FUNCTION_BLOCK FB_CRYO_VALVE_CTRL EXTENDS FB_CRYO_BIN_CTRL
VAR_INPUT
END_VAR
VAR_OUTPUT
END_VAR
VAR
	//
	// Alarm handling
	//
	// List of alarms to be handled by Valve.
	// Alarms cannot be defined in FB_CRYO_BIN_CTRL,
	// because they are specific to the device/controller.
	// There are three alarms for Valves:
	//   0: NOT_OP
	//   1: CLOSE failed
	//   2: OPEN  failed
	arrEventEntry : ARRAY [0..2] OF TcEventEntry;
	// Alarm handler FB
	fbAlarmHandler : FB_AlarmHandler;
END_VAR

// This call just configures logs at the very start.
// Logging is done by explicit calls to M_LogInfo().
logs(in_sName := in_sName);


// Execute parent FB.
SUPER^();


// Update the status.
// This will handle alarms as well.
M_SetStatus(stat.nState);

METHOD M_Configure
VAR_INPUT
END_VAR
// Device specific implementation
// 
arrEventEntry[0] := Tc_Events.CryoValveEventClass.HardwareError;
arrEventEntry[1] := Tc_Events.CryoValveEventClass.FailureOpen;
arrEventEntry[2] := Tc_Events.CryoValveEventClass.FailureClose;


// A MUST !!!
stat.bConfigured	:= TRUE;
END_METHOD

//
// Overrides the same method in FB_CRYO_BIN_CTRL.
//
// Set labels for logging.
//	OPEN, CLOSE (for valves)
METHOD M_GetStateLabel : STRING
VAR_INPUT
	state:	E_CRYO_BIN_CTRL_STATE;
END_VAR
CASE state OF
	E_CRYO_BIN_CTRL_STATE.OFF:
		M_GetStateLabel	:= 'CLOSED';
	
	E_CRYO_BIN_CTRL_STATE.ACTIVE_SWITCHING_ON:
		M_GetStateLabel	:= 'OPENING...';
	
	E_CRYO_BIN_CTRL_STATE.ACTIVE_OFF:
		M_GetStateLabel	:= 'CLOSED';
	
	E_CRYO_BIN_CTRL_STATE.ACTIVE_ON:
		M_GetStateLabel	:= 'OPEN';
	
	E_CRYO_BIN_CTRL_STATE.ACTIVE_SWITCHING_OFF:
		M_GetStateLabel	:= 'CLOSING...';
	
	E_CRYO_BIN_CTRL_STATE.ERROR:
		M_GetStateLabel	:= 'ERROR';
END_CASE
END_METHOD

METHOD M_SetStatus
VAR_INPUT
	nState:	E_CRYO_BIN_CTRL_STATE;
END_VAR
// Execute the status of the parent FB.
SUPER^.M_SetStatus(nState);


// Handle alarms
M_UpdateAlarms();
END_METHOD

METHOD M_UpdateAlarms
VAR_INPUT
END_VAR
VAR
	stEventEntry : TcEventEntry;
	sText : STRING;
END_VAR
// Array of EventEntry is initialised in the M_Configure method with 
// the alarms defined for the Valve.

fbAlarmHandler(stAlarms := stat.stAlarms);


// Trigger alarms in case of failure.
// The alarms are raised with a rising edge trigger.
// The alarms are cleared with a falling edge trigger.
IF stat.nState = E_CRYO_BIN_CTRL_STATE.ERROR THEN
	IF Actuator.i_nCouplerState <> 8 THEN
		// System not OPERATIONAL or
		// i_nCouplerState not linked to State variable.
		fbAlarmHandler.M_SetAlarm(Tc_Events.CryoValveEventClass.HardwareError);
		stat.sState	:= 'ERROR: System not OPERATIONAL';
	ELSIF Actuator.stat.nLastCommand = E_CRYO_BIN_ACT_CMD.OFF	THEN
		// Valve failed to Close.
		fbAlarmHandler.M_SetAlarm(Tc_Events.CryoValveEventClass.FailureClose);
		stat.sState	:= 'ERROR: Valve failed to CLOSE.';
	ELSIF Actuator.stat.nLastCommand = E_CRYO_BIN_ACT_CMD.ON	THEN
		// Valve failed to Open.
		fbAlarmHandler.M_SetAlarm(Tc_Events.CryoValveEventClass.FailureOpen);
		stat.sState	:= 'ERROR: Valve failed to OPEN.';
	END_IF

END_IF

//
// Clear non-active alarms
// Alarms and their indexes are defined in M_Configure().
// There are three alarms for Valves:
//   0: NOT_OP
//   1: CLOSE failed
//   2: OPEN  failed
//
IF fbAlarmHandler.arrAlarmState[0]  AND  Actuator.i_nCouplerState = 8 THEN
	fbAlarmHandler.M_ClearAlarm(Tc_Events.CryoValveEventClass.HardwareError);
END_IF

IF fbAlarmHandler.arrAlarmState[1]  AND  stat.nState <> E_CRYO_BIN_CTRL_STATE.ERROR THEN
	fbAlarmHandler.M_ClearAlarm(Tc_Events.CryoValveEventClass.FailureClose);
END_IF

IF fbAlarmHandler.arrAlarmState[2] = TRUE  AND  stat.nState <> E_CRYO_BIN_CTRL_STATE.ERROR THEN
	fbAlarmHandler.M_ClearAlarm(Tc_Events.CryoValveEventClass.FailureOpen);
END_IF


fbAlarmHandler.M_ProcessAlarms(
	arrEventEntry := arrEventEntry,
	sEventString := in_sName);
END_METHOD

METHOD M_User_SetAction : INT
VAR_INPUT
END_VAR
// TODO USER
// Set Valve command based on the input parameter in_bEnable.
//
	
IF	stat.nState = E_CRYO_BIN_CTRL_STATE.ACTIVE_OFF  AND in_bEnable THEN
	// Activate the actuator, i.e. open the valve
	M_User_SetAction	:= E_CRYO_BIN_CTRL_ACTION.ON;
ELSIF  stat.nState = E_CRYO_BIN_CTRL_STATE.ACTIVE_ON AND NOT in_bEnable THEN
	// Dectivate the actuator, i.e. close the valve
	M_User_SetAction	:= E_CRYO_BIN_CTRL_ACTION.OFF;
ELSE
	// Don't do anything
	M_User_SetAction	:= E_CRYO_BIN_CTRL_ACTION.NONE;
END_IF
END_METHOD

END_FUNCTION_BLOCK

(* stored: Version 1.1.0.1, ProductVersion 3.1.4024.14
   POU FB_CRYO_VALVE_CTRL: Id {821ef5cb-5c3c-4548-8cdd-f457c89df676}, SpecialFunc None
   Method M_Configure: Id {575769a3-a950-43a6-baea-8fe18b9cc362}
   Method M_GetStateLabel: Id {6a029015-f860-4667-b045-190dc1159f0d}
   Method M_SetStatus: Id {4aedb583-a641-44e2-9926-6d1ee3abadf1}
   Method M_UpdateAlarms: Id {2d0c7459-e7b0-4922-a181-0aa4996638a1}
   Method M_User_SetAction: Id {60abe389-4ad1-49f5-a9ed-250397cb9229} *)
